(* PLC project To_FTP_server, Beckhoff Automation GmbH TwinCAT PLC Control 3.5.13.20 *)
(* stored: creationDateTime 2020-09-10T09:39:55.3277713, modificationDateTime 2020-09-10T09:39:55.3357488 *)

FUNCTION_BLOCK FB_Upload_ToServer
VAR_INPUT
	bStartstop 			: BOOL;
	sHost :STRING;
	sUsername:STRING:='FTPclient';
	sPassword:STRING:= 'Fabslog8721';
	sSrcFile:STRING:= '\FTPclient\out\TestToServer.txt';
	sDesFile:STRING:= '\in\TestFromClient.txt';
END_VAR
VAR_OUTPUT
	err 				: BOOL;
	errid 				: UDINT;
END_VAR
VAR
	RisingEdge 			: R_TRIG;
	
	state				: BYTE;
	fbFTP_Open1 		: FB_FTP_OpenEX;
	fbFTPFileUpload1: FB_FTP_FileUpload;
	fbFTP_Close1 		: FB_FTP_Close;
	busy 				: BOOL;

	handle 				: T_HFTP;
	progress 			: UDINT;

END_VAR

            RisingEdge(CLK:= bStartstop);
IF RisingEdge.Q THEN
	state := 1;
END_IF

CASE state OF
	0:
		;

	1:
		fbFTP_Open1(
			sNetID:= ,
			sHost:= sHost ,
			nPort:= 21,
			sUsername:= sUsername,
	        sPassword:= sPassword,
			bExecute:= TRUE,
			tTimeout:= T#15S,
			 eMode    := 0,
			bBusy=> busy,
			bError=> err,
			nErrId=> errid,
			hFTP=> handle);

		IF NOT busy AND NOT err THEN
			fbFTP_Open1(bExecute:= FALSE);
			state := 2;
			
		END_IF

	2:
		fbFTPFileUpload1(
	sNetID:='' ,
     hFTP:=handle,
	sSrcFile:= sSrcFile,
	sDesFile:=sDesFile,
	bExecute:= TRUE,
	tTimeout:= T#15s,
	bBusy=> busy,
	bError=> err,
	nErrId=> errid,
	nProgress=> progress);

		IF NOT busy AND NOT err THEN
			fbFTPFileUpload1(bExecute:= FALSE);
			state := 3;
		END_IF

	3:
		fbFTP_Close1(
			sNetID:= ,
			hFTP:= handle,
			bExecute:= TRUE,
			tTimeout:= T#15s,
			bBusy => busy,
			bError => err,
			nErrId => errid);

		IF NOT busy AND NOT err THEN
			fbFTP_Close1(bExecute:= FALSE);
			state := 0;
		END_IF

END_CASE
          
END_FUNCTION_BLOCK
